FUNCTION_BLOCK FB_MruInterface
VAR_INPUT
END_VAR
VAR_OUTPUT
	feedback : ST_FeedbackMru;
	active : BOOL := FALSE;
END_VAR
VAR
	// Udp related
	udpServer : FB_UdpServerRT(0, 0, 0, 0, 0); // Dummy constructor
	
	{attribute 'tc_no_symbol'}
	rxUdpBE : ST_RxUdpMru;
	{attribute 'tc_no_symbol'}
	rxUdp : ST_RxUdpMru;
	
	// Hmi connection
	pTxHmi : POINTER TO ST_TxHmiMru;
	
	// Actviity monitoring
	frame : DINT := 0;
	frameOld : DINT := 0;
	frameLoss : DINT := 0;
END_VAR

// Check activity
frame := rxUdp.SystemTime;
IF frame <> frameOld THEN
	// Update frame old
	frameOld := frame;
	
	// Reset frameLoss
	frameLoss := 0;
ELSE
	// Count frame losses
	frameLoss := frameLoss + 1;
END_IF

// Set activity status after 1 second given 5ms in ms
IF frameLoss > 200 THEN
	active := FALSE;
ELSE
	active := TRUE;
END_IF

// Update udpServer
udpServer();

// Swap byte order on all float variables
rxUdp := BigToLittleEndian(rxUdpBE);

// ### Feedback ###
// E-Motion Body fixed positions
feedback.eta[0] := rxUdp.PosCg_F;
feedback.eta[1] := rxUdp.PosCg_S;
feedback.eta[2] := rxUdp.PosCg_D;
feedback.eta[3] := rxUdp.Roll;
feedback.eta[4] := rxUdp.Pitch;
feedback.eta[5] := rxUdp.Yaw;

// E-Motion Body fixed velocites
feedback.v[0] := rxUdp.VelCg_F;
feedback.v[1] := rxUdp.VelCg_S;
feedback.v[2] := rxUdp.VelCg_D;
feedback.v[3] := rxUdp.AngRate_R;
feedback.v[4] := rxUdp.AngRate_P;
feedback.v[5] := rxUdp.AngRate_Y;

// Update HMI Data
UpdateHMI();

METHOD BigToLittleEndian : ST_RxUdpMru 
VAR_INPUT
	rxUdpBE : ST_RxUdpMru;
END_VAR
VAR
	nData : UINT;
	n : UINT;
	pOffset : UINT;
	bytesBE : ARRAY [0..3] OF BYTE;
	bytesLE : ARRAY [0..3] OF BYTE;
	
	rxUdpLE : ST_RxUdpMru;
END_VAR
// NOTE: Only works with ST_RxMru struct!!! Not a genral function

nData := SIZEOF(rxUdpBE);

FOR n := 0 TO (nData/4 - 2) DO
	// Current pointer offset index
	pOffset := 3 + 4*n;

	IF pOffset <= nData THEN
		MEMCPY(ADR(bytesBE), ADR(rxUdpBE) + pOffset, 4);
	
		// Swap bytes from BE -> LE
		bytesLE[3] := bytesBE[0];
		bytesLE[2] := bytesBE[1];
		bytesLE[1] := bytesBE[2];
		bytesLE[0] := bytesBE[3];
		
		MEMCPY(ADR(rxUdpLE) + pOffset, ADR(bytesLE), 4);
	END_IF
END_FOR

BigToLittleEndian := rxUdpLE;
END_METHOD

METHOD FB_exit : BOOL
VAR_INPUT
	bInCopyCode : BOOL; // if TRUE, the exit method is called for exiting an instance that is copied afterwards (online change).
END_VAR
END_METHOD

METHOD FB_init : BOOL
VAR_INPUT
	bInitRetains : BOOL; // if TRUE, the retain variables are initialized (warm start / cold start)
	bInCopyCode : BOOL;  // if TRUE, the instance afterwards gets moved into the copy code (online change)
	
	// Init variables
	localPort : UINT;
	_pTxHmi : POINTER TO ST_TxHmiMru;
END_VAR
pTxHmi := _pTxHmi;

// Initilize the udpServer
udpServer.FB_init(
	bInitRetains,
	bInCopyCode,
	localPort,
	SIZEOF(rxUdpBE),
	ADR(rxUdpBE),
	0,
	0
);
END_METHOD

METHOD FB_reinit : BOOL
VAR_INPUT
END_VAR
END_METHOD

METHOD UpdateHMI
VAR_INPUT
END_VAR
VAR
	i : UINT;
END_VAR
// Update global Hmi data
IF active THEN
	pTxHmi^.status := 0;
ELSE
	pTxHmi^.status := -1;
END_IF

// Set MRU feedback
FOR i := 0 TO 5 DO
	pTxHmi^.eta[i] := LREAL_TO_REAL(feedback.eta[i]);
END_FOR
END_METHOD

END_FUNCTION_BLOCK

(* stored: Version 1.1.0.1, ProductVersion 3.1.4022.18
   POU FB_MruInterface: Id {c6b5539c-66b4-48be-8e8d-e330098c72f8}, SpecialFunc None
   Method BigToLittleEndian: Id {55be5d21-786e-44c3-a382-2ff80affc77c}
   Method FB_exit: Id {a3e9d2a2-7999-4f51-bfdc-9869126d272a}
   Method FB_init: Id {3130c499-1695-4075-b5a0-733165c80fd1}
   Method FB_reinit: Id {1faf6911-8283-46ae-9bd2-81f20ae258ae}
   Method UpdateHMI: Id {3ac8500f-b565-43be-93ea-37942fa30b65} *)
